ABB RobotStudio station: station_external_mechanism.rspag

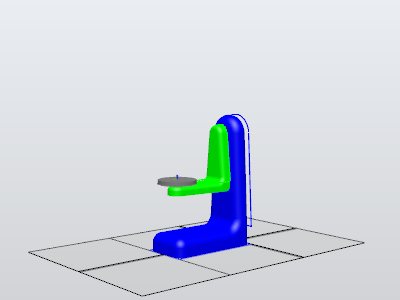
Station Station (saved by RobotStudio 24.1.10713.1)
Layout (positions relative to the parent item):
  - External_Mechanism [mechanism, from Module 3\External_Mechanism.rslib] at (0, 0, 0) mm; joint values [0, 0] (rad or m)
